TYPE CreateDirBusy :
UNION
	stCreateDirBusy : ST_CreateDirBusy;
	bitCalculator : BYTE;
END_UNION
END_TYPE

(* stored: Version 1.1.0.1, ProductVersion 3.1.4024.12
   DUT CreateDirBusy: Id {66e1fbf2-9013-4358-a478-b86967256d28} *)
